FUNCTION_BLOCK GraphFactory IMPLEMENTS I_GraphFactory
VAR
	nodePrototypes : NodePrototypes;
END_VAR

METHOD PUBLIC Accept
VAR_INPUT
	Visitor : I_GraphFactoryVisitor;
END_VAR
Visitor.VisitTcGraph(this^);
END_METHOD

METHOD PUBLIC Create : I_Graph
VAR
	pGraph : POINTER TO Graph;
END_VAR
pGraph := __NEW(Graph(NodePrototypes := THIS^.nodePrototypes));
Create := pGraph^;
END_METHOD

METHOD PUBLIC GetNodePrototypes : I_NodePrototypes
VAR_INPUT
END_VAR
GetNodePrototypes := nodePrototypes;
END_METHOD

METHOD PUBLIC InstallNodePack
VAR_INPUT
	NodePack : I_NodePack;
END_VAR
NodePack.RegisterWithGraph(This^);
END_METHOD

METHOD PUBLIC RegisterNodeByType
VAR_INPUT
	NodeType : T_MAXSTRING;
	NodePrototype : I_NodePrototype;	
END_VAR
nodePrototypes.InsertByType(NodeType,NodePrototype);
END_METHOD

METHOD PUBLIC SerializeWith
VAR_INPUT
	Serializer : I_Serializer;
END_VAR
Serializer.StartObject();
Serializer.Addkey('registeredNodes');
Serializer.AddObject(nodePrototypes);
Serializer.EndObject();
END_METHOD

END_FUNCTION_BLOCK

(* stored: Version 1.1.0.1, ProductVersion 3.1.4024.12
   POU GraphFactory: Id {3cf4dffb-2e67-0cde-05c3-0b7a44e6e216}, SpecialFunc None
   Method Accept: Id {d8350354-5d0e-015a-02f7-c388e7f54195}
   Method Create: Id {3dacf3c5-2186-0d1e-08e0-d29f6557f3d4}
   Method GetNodePrototypes: Id {4c05128d-a009-43a5-a61e-a66570dfd201}
   Method InstallNodePack: Id {0ec00c43-b35f-0669-2893-bc57927b1baa}
   Method RegisterNodeByType: Id {e69125b8-4a8c-01f5-3b08-4f76913c652b}
   Method SerializeWith: Id {198adf2e-d702-4dee-bba8-c3eb7ef16e84} *)
